FUNCTION_BLOCK CSVWriter IMPLEMENTS ITF_Writer
VAR
END_VAR

METHOD WriteMessage : BOOL
VAR_INPUT
	SomeString	: STRING(80);
END_VAR
ADSLOGSTR(msgCtrlMask := ADSLOG_MSGTYPE_LOG, msgFmtStr := 'I wrote a CSV line with: %s',strArg := SomeString);
END_METHOD

END_FUNCTION_BLOCK

(* stored: Version 1.1.0.1, ProductVersion 3.1.4024.12
   POU CSVWriter: Id {c850e885-e42f-4ca8-a387-23343dec58d0}, SpecialFunc None
   Method WriteMessage: Id {fbd2ee40-6875-45ff-a00d-2137b7064d42} *)
